				(* If no error, read one page of historical data *)
				FaultData.AlarmID 		:= ModBus.MB_Resp.Data[0];
				FaultData.SuppTime 		:= BUILD_16TO32_COPY(ModBus.MB_Resp.Data[1],ModBus.MB_Resp.Data[2]);
				FaultData.OpTime 		:= BUILD_16TO32_COPY(ModBus.MB_Resp.Data[3],ModBus.MB_Resp.Data[4]);
				FaultData.InvStatus 	:= ModBus.MB_Resp.Data[5];
				FaultData.Vpv_ref 		:= ModBus.MB_Resp.Data[6];
				FaultData.Vpv 			:= ModBus.MB_Resp.Data[7];
				FaultData.Vmain 		:= ModBus.MB_Resp.Data[8];
				FaultData.Status2 		:= ModBus.MB_Resp.Data[9];
				FaultData.Status1 		:= ModBus.MB_Resp.Data[10];
				FaultData.Tboard 		:= ModBus.MB_Resp.Data[11];
				FaultData.Tigbt 		:= ModBus.MB_Resp.Data[12];
				FaultData.I_u 			:= ModBus.MB_Resp.Data[13];
				FaultData.I_v 			:= ModBus.MB_Resp.Data[14];
				FaultData.I_w 			:= ModBus.MB_Resp.Data[15];
				FaultData.ClampStatus 	:= ModBus.MB_Resp.Data[16];
				FaultData.DigOutput 	:= ModBus.MB_Resp.Data[17];
				FaultData.IgbtFault 	:= ModBus.MB_Resp.Data[18];
				FaultData.Psupp			:= BUILD_16TO32_COPY(ModBus.MB_Resp.Data[19],ModBus.MB_Resp.Data[20]);
				FaultData.Epv 			:= BUILD_16TO32_COPY(ModBus.MB_Resp.Data[22],ModBus.MB_Resp.Data[23]);

				ModBus.MB_Lock := FALSE;		(* All 8 pages transmitted *)
				FaultAddr 	:= 0;				(* Reset start address *)
				state_fault := WAIT_STATE;
				last_state	:= WAIT_STATE;
				retry := 0;		(* Reset retry counter *)
		
			END_IF
		END_IF

	ERROR_STATE:

		IF retry>3 THEN
			IF NOT ModBus.MB_Lock THEN LogEv(EL_Alarm,EO_INV,ID,5,'');						(* ModBus not free	*)
			ELSE LogEv(EL_Alarm,EO_INV,ID,4,SEL(ModBus.MB_MASTER.MB_Error<>0,'0','1'));		(* ModBus communication error *)
			END_IF

			FaultAddr 	:= 0;
			state_fault := WAIT_STATE;
		ELSE
			retry := retry + 1;
			state_fault := last_state;
		END_IF
END_CASE
END_ACTION

(* POU Plant_Objects/obj_MODBUS_STR_ES889, ST *)
FUNCTION_BLOCK obj_MODBUS_STR_ES889
(* === MODBUS SMART STRING BOX ES889 ===
   v1.0[15/06/15] - Versioning
*)
VAR CONSTANT
		WAIT_STATE		:	BYTE := 0;
		QUERY_MEAS_1	:	BYTE := 1;
		QUERY_MEAS_2	:	BYTE := 2;
		QUERY_MASK		:	BYTE := 3;
		QUERY_PANELS	:	BYTE := 4;
		END_READ		:	BYTE := 5;

		QUERY_FAULT_LIST:	BYTE := 10;
		LOG_HISTORICAL	:	BYTE := 11;

		ERROR_STATE		:	BYTE := 100;

END_VAR
VAR_INPUT
		ID			:	BYTE;				(* Logical device ID needed for Clevergy purpose and log	*)
		Address		:	BYTE;				(* Modbus address of the device	*)

		RefreshTime	: 	TIME := T#1m;

		(* Read fault list *)
		FaultAddr	:	WORD;

		retryErrMax	:	BYTE := 15;		(* 15 minutes *)
END_VAR
VAR_IN_OUT
		ModBus		: obj_MODBUS;
END_VAR
VAR_OUTPUT
		Status_Log	: BYTE;
		Status_Vis	: DWORD;
END_VAR
VAR
		InitOK		: BOOL;			(* Flag that indicates if the VARS have been initialized or not	*)

		Data		: typ_MODBUS_STR_ES889;
		tempData	: typ_MODBUS_STR_ES889;
		FaultData	: typ_MODBUS_STR_ES889_His;

		(* Modbus State machine variables	*)
		state		:	BYTE;
		state_fault	:	BYTE;
		last_state	:	BYTE;
		retry		:	BYTE;
		retryErr	:	BYTE;
		ReadTmr		:	TON := (PT:=t#5s);
		fModbusAlr	:	BOOL;

		counter		:	BYTE;

		Alarm		: FLT_EVENT;
		WrnPerform	: FLT_EVENT;
		ModbusAlr	: FLT_EVENT := (INITEV:=FALSE);

		ActualAlarm	: BYTE;
		OldAlarm	: BYTE;
		ActualStolen: WORD;
		OldStolen	: WORD;
		OldOpen		: WORD;
		PerformWrn	: WORD;
		OldPerform	: WORD;

		AlarmCtr	: BYTE;
		WarningCtr	: BYTE;

		s1			: STRING;

		fTimeout	: BOOL;
END_VAR
IF NOT InitOK THEN
	ReadTmr.PT := WORD_TO_TIME((Plant_INV+ID)*2000);
	InitOK := TRUE;
END_IF

IF FaultAddr=0 THEN

	Stm();

	(**** Check String Box ALARM ****)
	CheckAlarm();

ELSE

	StmFault();

END_IF

(* Set "Status_Log" according to actual object status	*)
IF AlarmCtr > 0 THEN
	Status_Log := 2;
	Status_Vis := COLOR_RED;
ELSIF WarningCtr > 0 THEN
	Status_Log := 1;
	Status_Vis := COLOR_YELLOW;
ELSE
	Status_Log := 0;
	Status_Vis := COLOR_GREEN;
END_IF
END_FUNCTION_BLOCK
ACTION AddLogData:
Logger.s1:=INSERT('&STR=',BYTE_TO_STRING(ID),4);
IF ID<10 THEN Logger.s1:=INSERT(Logger.s1,'0',4); END_IF

(* Create messagge to append to the log file in string format, containing the historical value for current alarm	*)
Logger.s1:=CONCAT(Logger.s1,WORD_TO_STRING(Data.Istring1));				Logger.s1:=CONCAT(Logger.s1,';');
Logger.s1:=CONCAT(Logger.s1,WORD_TO_STRING(Data.Istring2));				Logger.s1:=CONCAT(Logger.s1,';');
Logger.s1:=CONCAT(Logger.s1,WORD_TO_STRING(Data.Istring3));				Logger.s1:=CONCAT(Logger.s1,';');
Logger.s1:=CONCAT(Logger.s1,WORD_TO_STRING(Data.Istring4));				Logger.s1:=CONCAT(Logger.s1,';');
Logger.s1:=CONCAT(Logger.s1,WORD_TO_STRING(Data.Istring5));				Logger.s1:=CONCAT(Logger.s1,';');
Logger.s1:=CONCAT(Logger.s1,WORD_TO_STRING(Data.Istring6));				Logger.s1:=CONCAT(Logger.s1,';');
Logger.s1:=CONCAT(Logger.s1,WORD_TO_STRING(Data.Istring7));				Logger.s1:=CONCAT(Logger.s1,';');
Logger.s1:=CONCAT(Logger.s1,WORD_TO_STRING(Data.Istring8));				Logger.s1:=CONCAT(Logger.s1,';');
Logger.s1:=CONCAT(Logger.s1,WORD_TO_STRING(Data.Iavg));					Logger.s1:=CONCAT(Logger.s1,';');
Logger.s1:=CONCAT(Logger.s1,WORD_TO_STRING(Data.Imax));					Logger.s1:=CONCAT(Logger.s1,';');
Logger.s1:=CONCAT(Logger.s1,WORD_TO_STRING(Data.Imin));					Logger.s1:=CONCAT(Logger.s1,';');

Logger.s1:=CONCAT(Logger.s1,INT_TO_STRING(Data.Tboard));				Logger.s1:=CONCAT(Logger.s1,';');
Logger.s1:=CONCAT(Logger.s1,INT_TO_STRING(Data.Tenv));					Logger.s1:=CONCAT(Logger.s1,';');

Logger.s1:=CONCAT(Logger.s1,WORD_TO_STRING(Data.M019));					Logger.s1:=CONCAT(Logger.s1,';');
Logger.s1:=CONCAT(Logger.s1,WORD_TO_STRING(PerformWrn));				Logger.s1:=CONCAT(Logger.s1,';');

(* Add log returned by the object	*)
Logger.s1:=CONCAT(Logger.s1,BYTE_TO_STRING(Status_Log));

(* Add the entire new string "s1" with the updated measurements to the one has to be transmitted	*)
ADDSTRING(ADR(Logger.TData), ADR(Logger.s1), Logger.TLen);
END_ACTION
ACTION AppendMeasure:
(* Used to add signifcant measurements when an alarm happens (it's a sort of historical fault list, as described at page 40
   of the Programming Manual; the only difference is that is not used the one of the string box, but it's rebuild with the
   read measurements *)
s1 := CONCAT(s1,';');
s1 := CONCAT(s1, WORD_TO_STRING(SHR(Data.M018,8)));	(* Stolen string *)
s1 := CONCAT(s1,';');
s1 := CONCAT(s1, WORD_TO_STRING(Data.M019));		(* Open string *)
s1 := CONCAT(s1,';');
s1 := CONCAT(s1, INT_TO_STRING(Data.Tboard));		(* Board temperature *)
s1 := CONCAT(s1,';');
s1 := CONCAT(s1, DWORD_TO_STRING(Data.SuppTime));	(* Supply time *)
s1 := CONCAT(s1,';');
s1 := CONCAT(s1, DWORD_TO_STRING(Data.OpTime));		(* Operation time *)
END_ACTION
ACTION CheckAlarm:
(* Verify ModBus error	*)
ModbusAlr(IN:=fModbusAlr);

IF ModbusAlr.EVH THEN
	LogEv(EL_Alarm,EO_STR,ID,4,SEL(ModBus.MB_MASTER.MB_Error<>0,'0','1'));
	AlarmCtr := AlarmCtr + 1;
END_IF

IF ModbusAlr.EVL THEN
	LogEv(EL_Log,EO_STR,ID,9,'');
	AlarmCtr := SEL(AlarmCtr=0, AlarmCtr-1, 0);
END_IF


(* Verify StringBox error/alarm	*)
ActualAlarm := WORD_TO_BYTE(Data.M018 AND 16#0F);

Alarm(IN:=(ActualAlarm <> OldAlarm));

IF Alarm.EVH THEN
	IF ActualAlarm = 0 THEN
		AlarmCtr := SEL(AlarmCtr=0, AlarmCtr-1, 0);
	ELSE
		(* Alarm codes 8 and 9 are yet checked with open and stolen string dedicated filters *)
		IF ActualAlarm<8 AND ActualAlarm>9 THEN
			LogEv(EL_Alarm,EO_STR,ID,3,BYTE_TO_STRING(ActualAlarm));
			AppendMeasure();
			AlarmCtr := AlarmCtr + 1;
		END_IF
	END_IF

	OldAlarm := ActualAlarm;
END_IF

(**** Check if another string has been stolen ****)
ActualStolen := (SHR(Data.M018,8) AND 16#00FF);

IF ActualStolen <> OldStolen THEN
	IF ActualStolen = 0 THEN
		AlarmCtr := SEL(AlarmCtr=0, AlarmCtr-1, 0);
	ELSE
		LogEv(EL_Alarm,EO_STR,ID,6,WORD_TO_STRING(ActualStolen));
		AlarmCtr := AlarmCtr + 1;
	END_IF

	OldStolen := ActualStolen;
END_IF
END_ACTION
ACTION Stm:
CASE state OF

	WAIT_STATE:	(* Refresh time manager *)

		ReadTmr(IN:=NOT(ReadTmr.Q));
		IF ReadTmr.Q THEN

			ReadTmr.PT := RefreshTime;			(* Refresh timer range *)

			(* Reset state machine variables and counters *)
			retry	:= 0;
			counter := 0;
			last_state	:= WAIT_STATE;

			(* Start state machine	*)
			state := QUERY_MEAS_1;

		END_IF


	QUERY_MEAS_1:	(* External energy counters *)
		IF NOT ModBus.MB_Start AND (NOT ModBus.MB_Lock OR retry>0) THEN
			ModBus.MB_Lock := TRUE;
			ModBus.MB_Obj := EO_STR;
			ModBus.MB_ObjId := ID;

			ModBus.MB_Query.SlaveAddress := Address;
			ModBus.MB_Query.FunctionCode := 16#3;
			ModBus.MB_Query.Read_StartAddress := 1651;
			ModBus.MB_Query.Read_Quantity := 20;
			ModBus.MB_Start := TRUE;

			state := QUERY_MEAS_2;
		END_IF

	QUERY_MEAS_2:	(* Energy supplied to the net *)

		IF NOT ModBus.MB_Start THEN
			IF ModBus.MB_MASTER.bInterfaceError<>0 OR ModBus.MB_MASTER.MB_Error<>0 THEN
				last_state := QUERY_MEAS_1;
				state := ERROR_STATE;
			ELSE

				tempData.Istring1		:= ModBus.MB_Resp.Data[0];
				tempData.Istring2		:= ModBus.MB_Resp.Data[1];
				tempData.Istring3		:= ModBus.MB_Resp.Data[2];
				tempData.Istring4		:= ModBus.MB_Resp.Data[3];
				tempData.Istring5		:= ModBus.MB_Resp.Data[4];
				tempData.Istring6		:= ModBus.MB_Resp.Data[5];
				tempData.Istring7		:= ModBus.MB_Resp.Data[6];
				tempData.Istring8		:= ModBus.MB_Resp.Data[7];
				tempData.Iavg			:= ModBus.MB_Resp.Data[8];
				tempData.Imax			:= ModBus.MB_Resp.Data[9];
				tempData.Imin			:= ModBus.MB_Resp.Data[10];

				tempData.Radiation_h	:= ModBus.MB_Resp.Data[11];
				tempData.Radiation_m	:= ModBus.MB_Resp.Data[12];
				tempData.Tmodule		:= WORD_TO_INT(ModBus.MB_Resp.Data[13]);
				tempData.Tenv			:= WORD_TO_INT(ModBus.MB_Resp.Data[14]);
				tempData.Vwind			:= ModBus.MB_Resp.Data[15];
				tempData.Tboard			:= WORD_TO_INT(ModBus.MB_Resp.Data[16]);

				tempData.M018			:= ModBus.MB_Resp.Data[17];
				tempData.M019			:= ModBus.MB_Resp.Data[18];
				tempData.M020			:= ModBus.MB_Resp.Data[19];

				ModBus.MB_Query.SlaveAddress := Address;
				ModBus.MB_Query.FunctionCode := 16#3;
				ModBus.MB_Query.Read_StartAddress := 57;
				ModBus.MB_Query.Read_Quantity := 4;
				ModBus.MB_Start := TRUE;

				state := QUERY_MASK;
			END_IF
		END_IF

	QUERY_MASK:
		IF NOT ModBus.MB_Start THEN
			IF ModBus.MB_MASTER.bInterfaceError<>0 OR ModBus.MB_MASTER.MB_Error<>0 THEN
				last_state := QUERY_MEAS_2;
				state := ERROR_STATE;
			ELSE

				tempData.SuppTime	:= BUILD_16TO32_COPY(ModBus.MB_Resp.Data[0],ModBus.MB_Resp.Data[1]);
				tempData.OpTime		:= BUILD_16TO32_COPY(ModBus.MB_Resp.Data[2],ModBus.MB_Resp.Data[3]);

				ModBus.MB_Query.SlaveAddress := Address;
				ModBus.MB_Query.FunctionCode := 16#3;
				ModBus.MB_Query.Read_StartAddress := 250;
				ModBus.MB_Query.Read_Quantity := 2;
				ModBus.MB_Start := TRUE;

				state := QUERY_PANELS;

			END_IF
		END_IF

	QUERY_PANELS:
		IF NOT ModBus.MB_Start THEN
			IF ModBus.MB_MASTER.bInterfaceError<>0 OR ModBus.MB_MASTER.MB_Error<>0 THEN
				last_state := QUERY_MASK;
				state := ERROR_STATE;
			ELSE

				tempData.Mask	:= ModBus.MB_Resp.Data[0];

				ModBus.MB_Query.SlaveAddress := Address;
				ModBus.MB_Query.FunctionCode := 16#3;
				ModBus.MB_Query.Read_StartAddress := 294;
				ModBus.MB_Query.Read_Quantity := 1;
				ModBus.MB_Start := TRUE;

				state := END_READ;

			END_IF
		END_IF

	END_READ:

		IF NOT ModBus.MB_Start THEN
			IF ModBus.MB_MASTER.bInterfaceError<>0 OR ModBus.MB_MASTER.MB_Error<>0 THEN
				last_state := QUERY_PANELS;
				state := ERROR_STATE;
			ELSE
				tempData.Panels	:= ModBus.MB_Resp.Data[0];

				(* Copy temporary data *)
				MEMCPY(ADR(tempData), ADR(Data), SIZEOF(Data));
				PerformWrn := Data.M020 AND 16#00FF;

				fModbusAlr := FALSE;
				retryErr := 0;
				ModBus.MB_Lock := FALSE;
				state := WAIT_STATE;

				(*** TEST ***)
				fTimeout := FALSE;

			END_IF
		END_IF

	ERROR_STATE:	(* Error state *)

		IF retry < 3 THEN
			retry := retry+1;
			state := last_state;

		ELSE
			ModBus.MB_Lock := FALSE;

			(* Verify if slave is dead *)
			IF retryErr < retryErrMaX THEN
				retryErr := retryErr + 1;
			ELSE
				fModbusAlr := TRUE;
			END_IF

			state := WAIT_STATE;

			(*** TEST ***)
			fTimeout := TRUE;
		END_IF


		IF ModBus.MB_MASTER.MB_Error=MB_TIME_OUT AND ID<>10 THEN
			state := state;
		END_IF
ELSE
	state := WAIT_STATE;
END_CASE
END_ACTION
ACTION StmFault:
(* State machine *)
CASE state OF

	WAIT_STATE:
		IF NOT (ModBus.MB_Lock OR ModBus.MB_Start) THEN
			ModBus.MB_Lock := TRUE;
			counter := 0;
			retry 	:= 0;
			last_state  := WAIT_STATE;
			state_fault := QUERY_FAULT_LIST;
		ELSE
			last_state  := WAIT_STATE;
			state_fault := ERROR_STATE;
		END_IF

	QUERY_FAULT_LIST:
		ModBus.MB_Query.SlaveAddress := Address;
		ModBus.MB_Query.FunctionCode := 16#3;
		ModBus.MB_Query.Read_StartAddress := FaultAddr;
		ModBus.MB_Query.Read_Quantity := 7;
		ModBus.MB_Start := TRUE;

		state := END_READ;


	END_READ:
		IF NOT ModBus.MB_Start THEN
			IF ModBus.MB_MASTER.bInterfaceError <> 0 OR ModBus.MB_MASTER.MB_Error<>0 THEN
				(* If no error, read one page of historical data *)
				FaultData.M018	 		:= ModBus.MB_Resp.Data[0];
				FaultData.M020			:= ModBus.MB_Resp.Data[1];
				FaultData.Tmodule		:= WORD_TO_INT(ModBus.MB_Resp.Data[2]);
				FaultData.SuppTime		:= BUILD_16TO32_COPY(ModBus.MB_Resp.Data[3],ModBus.MB_Resp.Data[4]);
				FaultData.OpTime		:= BUILD_16TO32_COPY(ModBus.MB_Resp.Data[5],ModBus.MB_Resp.Data[6]);


				(* Send data to server	*)
				LogEv(EL_Evt,EO_STR,ID,9,s1);

				IF counter > 7 THEN
					ModBus.MB_Lock := FALSE;		(* All 8 pages transmitted *)
					FaultAddr 	:= 0;				(* Reset start address *)
					state_fault := WAIT_STATE;
					last_state	:= WAIT_STATE;
				ELSE
					state_fault := QUERY_FAULT_LIST;
				END_IF

				retry := 0;		(* Reset retry counter *)
			ELSE
				state := ERROR_STATE;
			END_IF
		END_IF

	ERROR_STATE:

		IF retry>3 THEN
			IF NOT ModBus.MB_Lock THEN LogEv(EL_Alarm,EO_STR,ID,5,'');						(* ModBus not free	*)
			ELSE LogEv(EL_Alarm,EO_STR,ID,4,SEL(ModBus.MB_MASTER.MB_Error<>0,'0','1'));		(* ModBus communication error *)
			END_IF

			FaultAddr 	:= 0;
			state_fault := WAIT_STATE;
		ELSE
			retry := retry + 1;
			state_fault := last_state;
		END_IF
END_CASE
END_ACTION

(* POU Utils Functions/PLANT_STATUS, ST *)
FUNCTION_BLOCK PLANT_STATUS
VAR_INPUT
	obj_Status		:	WORD;
END_VAR
VAR_OUTPUT
	plantStatus		:	WORD;
END_VAR
VAR
	Pwm				:	TON := (PT:=T#1s);
END_VAR
(*CASE plantStatus OF

	0:	(* Plant OK - Everything works well *)
		Pwm(IN:=FALSE);							(* Stop timer if running *)
		LAMP_AL := FALSE;						(* Keep the lamp switched off *)

	1:	(* Plant in warning *)
		Pwm(IN:= NOT(Pwm.Q));

		IF Pwm.Q THEN
			LAMP_AL := NOT LAMP_AL;				(* Toggle output *)
		END_IF

	2:	(* Plant in alarm *)
		Pwm(IN:=FALSE);							(* Stop timer if running *)
		LAMP_AL	:= TRUE;						(* Keep the lamp switched on *)

END_CASE*)

plantStatus := 0;		(* Reset plant status *)
END_FUNCTION_BLOCK
ACTION UpdateStatus:
IF plantStatus = 2 THEN

	RETURN;					(* If plant already in alarm condition do nothing *)

ELSE
	IF obj_Status <> 0 THEN
		plantStatus := obj_Status;			(* If plant in warning/normal condition and current object in alarm, update plant status *)
	END_IF
END_IF
END_ACTION

(* POU PLC_WDT_old, ST *)
FUNCTION PLC_WDT_old: DWORD VAR_INPUT dwEvent: DWORD; dwFilter: DWORD; dwOwner: DWORD; END_VAR
LogEv(EL_AlarmStop,EO_SYS,1,10,'Watchdog');
END_FUNCTION

(* POU Utils Functions/RAW16TOHEXSTR, ST *)
FUNCTION RAW16TOHEXSTR : STRING(128)
VAR_INPUT
	pData: POINTER TO BYTE;
	DataLen: BYTE;
END_VAR
VAR
	pt: POINTER TO BYTE;
	xl: BYTE;
END_VAR
pt:=ADR(RAW16TOHEXSTR);
xl:=0;

WHILE DataLen>0 AND xl<120 DO

	pData:=pData+1;

	pt^ := (pData^ / 16#10) + 48 + (((pData^ / 16#10)/10)*7);
	pt:=pt+1;
	pt^ := (pData^ AND 16#0F)  + 48 + (((pData^ AND 16#0F)/10)*7);
	pt:=pt+1;

	pData:=pData-1;

	pt^ := (pData^ / 16#10) + 48 + (((pData^ / 16#10)/10)*7);
	pt:=pt+1;
	pt^ := (pData^ AND 16#0F)  + 48 + (((pData^ AND 16#0F)/10)*7);
	pt:=pt+1;

	xl:=xl+4;

	DataLen:=DataLen-2;
	pData:=pData+2;

END_WHILE

pt^:=0;
END_FUNCTION

(* POU Utils Functions/RAWTOHEXSTR, ST *)
FUNCTION RAWTOHEXSTR : STRING(128)
VAR_INPUT
	pData: POINTER TO BYTE;
	DataLen: BYTE;
END_VAR
VAR
	pt: POINTER TO BYTE;
	xl: BYTE;
END_VAR
pt:=ADR(RAWTOHEXSTR);

xl:=2;

WHILE DataLen>0 AND xl<128 DO

	pt^ := (pData^ / 16#10) + 48 + (((pData^ / 16#10)/10)*7);
	pt:=pt+1;
	pt^ := (pData^ AND 16#0F)  + 48 + (((pData^ AND 16#0F)/10)*7);
	pt:=pt+1;

	xl:=xl+2;

	DataLen:=DataLen-1;
	pData:=pData+1;

END_WHILE

pt^:=0;
END_FUNCTION

(* POU Utils Functions/TONOF, ST *)
FUNCTION_BLOCK TONOF
VAR_INPUT
	IN		: BOOL;
	PT_ON	: TIME; (* time to pass, before OUT is set *)
	PT_OF	: TIME; (* time to pass, before OUT is reset *)
END_VAR
VAR_OUTPUT
	OUT		: BOOL;
END_VAR
VAR
	timer	: TON;
END_VAR
IF IN<>OUT THEN
	timer(IN:=TRUE,PT:=SEL(IN,PT_OF,PT_ON));
	IF timer.Q THEN OUT:=IN; END_IF
ELSE
	timer(IN:=FALSE);
END_IF
END_FUNCTION_BLOCK

(* Visualisation PLC_VISU
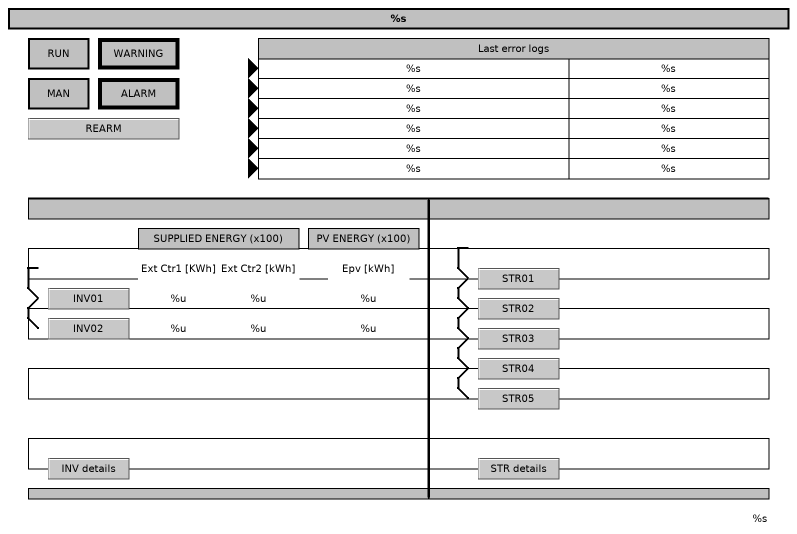
rectangle at (10,0)-(791,21): text "%s"; shows .Plant_NAME
rounded rectangle at (30,30)-(91,61): text "RUN"; alarm colour if NOT Mode_Manual; runs INTERN ASSIGN Mode_Manual:=(FALSE)
rounded rectangle at (30,70)-(91,101): text "MAN"; alarm colour if Mode_Manual; runs INTERN ASSIGN Mode_Manual:=(TRUE)
rectangle at (570,50)-(771,71): text "%s"; shows Sys.LastLogs_Msg[0]
polygon at (250,150)-(260,170): invisible if Sys.LastLogs_Idx<>0
rectangle at (570,70)-(771,91): text "%s"; shows Sys.LastLogs_Msg[1]
polygon at (250,50)-(260,70): invisible if Sys.LastLogs_Idx<>1
rectangle at (570,90)-(771,111): text "%s"; shows Sys.LastLogs_Msg[2]
polygon at (250,70)-(260,90): invisible if Sys.LastLogs_Idx<>2
rectangle at (570,110)-(771,131): text "%s"; shows Sys.LastLogs_Msg[3]
polygon at (250,90)-(260,110): invisible if Sys.LastLogs_Idx<>3
rectangle at (570,130)-(771,151): text "%s"; shows Sys.LastLogs_Msg[4]
polygon at (250,110)-(260,130): invisible if Sys.LastLogs_Idx<>4
rectangle at (570,150)-(771,171): text "%s"; shows Sys.LastLogs_Msg[5]
polygon at (250,130)-(260,150): invisible if Sys.LastLogs_Idx<>5
rectangle at (260,50)-(571,71): text "%s"; shows Sys.LastLogs_Dat[0]
rectangle at (260,70)-(571,91): text "%s"; shows Sys.LastLogs_Dat[1]
rectangle at (260,90)-(571,111): text "%s"; shows Sys.LastLogs_Dat[2]
rectangle at (260,110)-(571,131): text "%s"; shows Sys.LastLogs_Dat[3]
rectangle at (260,130)-(571,151): text "%s"; shows Sys.LastLogs_Dat[4]
rectangle at (260,150)-(571,171): text "%s"; shows Sys.LastLogs_Dat[5]
rectangle at (100,70)-(181,101): text "ALARM"; alarm colour if Sys.Alarm; runs INTERN ASSIGN Mode_Manual:=(FALSE)
rectangle at (100,30)-(181,61): text "WARNING"; alarm colour if Sys.Warning; runs INTERN ASSIGN Mode_Manual:=(TRUE)
button at (30,110)-(181,131): text "REARM"; runs INTERN ASSIGN Sys.Alarm:=(FALSE);INTERN ASSIGN Sys.Warning:=(FALSE)
button at (50,280)-(131,301): text "INV01"; runs INTERN ASSIGN INV[1].Cmd:=(0);INTERN ASSIGN INV[1].fRemoteCmd:=(TRUE)
rectangle at (260,30)-(771,51): text "Last error logs"
button at (50,310)-(131,331): text "INV02"; runs INTERN ASSIGN INV[2].Cmd:=(0);INTERN ASSIGN INV[2].fRemoteCmd:=(TRUE)
rectangle at (140,250)-(221,271): text "Ext Ctr1 [KWh]"
rectangle at (140,280)-(221,301): text "%u"; shows INV[1].Data.Esup_ExtCtr1
rectangle at (140,310)-(221,331): text "%u"; shows INV[2].Data.Esup_ExtCtr1
rounded rectangle at (140,220)-(301,241): text "SUPPLIED ENERGY (x100)"
button at (50,450)-(131,471): text "INV details"; opens PLC_VISU_INV
button at (480,260)-(561,281): text "STR01"; runs INTERN ASSIGN STR[1].Cmd:=(0);INTERN ASSIGN STR[1].fRead:=(TRUE)
button at (480,290)-(561,311): text "STR02"; runs INTERN ASSIGN STR[2].Cmd:=(0);INTERN ASSIGN STR[2].fRead:=(TRUE)
button at (480,320)-(561,341): text "STR03"; runs INTERN ASSIGN STR[3].Cmd:=(0);INTERN ASSIGN STR[3].fRead:=(TRUE)
button at (480,350)-(561,371): text "STR04"; runs INTERN ASSIGN STR[4].Cmd:=(0);INTERN ASSIGN STR[4].fRead:=(TRUE)
button at (480,380)-(561,401): text "STR05"; runs INTERN ASSIGN STR[5].Cmd:=(0);INTERN ASSIGN STR[5].fRead:=(TRUE)
button at (480,450)-(561,471): text "STR details"; opens PLC_VISU_STR
rectangle at (220,250)-(301,271): text "Ext Ctr2 [kWh]"
rectangle at (220,280)-(301,301): text "%u"; shows INV[1].Data.ExtCtr2
rectangle at (220,310)-(301,331): text "%u"; shows INV[2].Data.ExtCtr2
rounded rectangle at (310,220)-(421,241): text "PV ENERGY (x100)"
rectangle at (330,250)-(411,271): text "Epv [kWh]"
rectangle at (330,280)-(411,301): text "%u"; shows INV[1].Data.Epv
rectangle at (330,310)-(411,331): text "%u"; shows INV[2].Data.Epv
rectangle at (430,500)-(771,521): text "%s"; shows Sys.Time_LogString
15 more shapes without text or variables
9 elements of other kinds (tables, trends, ...) not read
*)

(* Visualisation PLC_VISU_INV
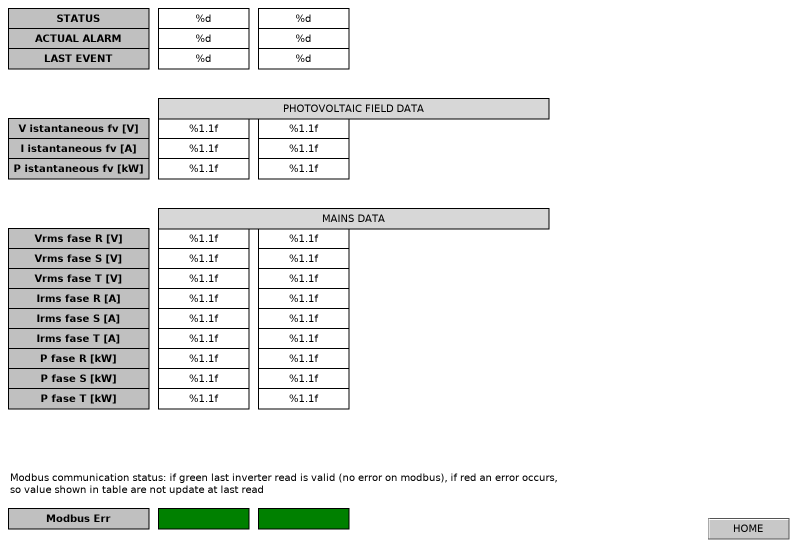
rectangle at (10,160)-(151,181): text "V istantaneous fv [V]"
rectangle at (10,180)-(151,201): text "I istantaneous fv [A]"
rectangle at (10,200)-(151,221): text "P istantaneous fv [kW]"
rectangle at (10,270)-(151,291): text "Vrms fase R [V]"
rectangle at (10,290)-(151,311): text "Vrms fase S [V]"
rectangle at (10,310)-(151,331): text "Vrms fase T [V]"
rectangle at (10,330)-(151,351): text "Irms fase R [A]"
rectangle at (10,350)-(151,371): text "Irms fase S [A]"
rectangle at (10,370)-(151,391): text "Irms fase T [A]"
rectangle at (10,390)-(151,411): text "P fase R [kW]"
rectangle at (10,410)-(151,431): text "P fase S [kW]"
rectangle at (10,430)-(151,451): text "P fase T [kW]"
rectangle at (10,50)-(151,71): text "STATUS"
rectangle at (10,70)-(151,91): text "ACTUAL ALARM"
rectangle at (160,160)-(251,181): text "%1.1f"; shows WORD_TO_REAL(.INV[1].Data.Vpv)/10
rectangle at (160,180)-(251,201): text "%1.1f"; shows WORD_TO_REAL(INV[1].Data.Ipv)/10
rectangle at (160,270)-(251,291): text "%1.1f"; shows WORD_TO_REAL(INV[1].Data.Vrms_r)/10
rectangle at (160,290)-(251,311): text "%1.1f"; shows WORD_TO_REAL(INV[1].Data.Vrms_s)/10
rectangle at (160,310)-(251,331): text "%1.1f"; shows WORD_TO_REAL(INV[1].Data.Vrms_t)/10
rectangle at (160,330)-(251,351): text "%1.1f"; shows INT_TO_REAL(INV[1].Data.Irms_r)/10
rectangle at (160,350)-(251,371): text "%1.1f"; shows INT_TO_REAL(INV[1].Data.Irms_s)/10
rectangle at (160,370)-(251,391): text "%1.1f"; shows INT_TO_REAL(INV[1].Data.Irms_t)/10
rectangle at (160,390)-(251,411): text "%1.1f"; shows INT_TO_REAL(INV[1].Data.P_r)/10
rectangle at (160,410)-(251,431): text "%1.1f"; shows INT_TO_REAL(INV[1].Data.P_s)/10
rectangle at (160,430)-(251,451): text "%1.1f"; shows INT_TO_REAL(INV[1].Data.P_t)/10
rectangle at (160,200)-(251,221): text "%1.1f"; shows INT_TO_REAL(INV[1].Data.Ppv)/10
rectangle at (160,50)-(251,71): text "%d"; shows INV[1].Data.Status
rectangle at (160,70)-(251,91): text "%d"; shows .INV[1].Data.ActiveAlarm
rectangle at (260,160)-(351,181): text "%1.1f"; shows WORD_TO_REAL(INV[2].Data.Vpv)/10
rectangle at (260,180)-(351,201): text "%1.1f"; shows WORD_TO_REAL(INV[2].Data.Ipv)/10
rectangle at (260,270)-(351,291): text "%1.1f"; shows WORD_TO_REAL(INV[2].Data.Vrms_r)/10
rectangle at (260,290)-(351,311): text "%1.1f"; shows WORD_TO_REAL(INV[2].Data.Vrms_s)/10
rectangle at (260,310)-(351,331): text "%1.1f"; shows WORD_TO_REAL(INV[2].Data.Vrms_t)/10
rectangle at (260,330)-(351,351): text "%1.1f"; shows INT_TO_REAL(INV[2].Data.Irms_r)/10
rectangle at (260,350)-(351,371): text "%1.1f"; shows INT_TO_REAL(INV[2].Data.Irms_s)/10
rectangle at (260,370)-(351,391): text "%1.1f"; shows INT_TO_REAL(INV[2].Data.Irms_t)/10
rectangle at (260,390)-(351,411): text "%1.1f"; shows INT_TO_REAL(INV[2].Data.P_r)/10
rectangle at (260,410)-(351,431): text "%1.1f"; shows INT_TO_REAL(INV[2].Data.P_s)/10
rectangle at (260,430)-(351,451): text "%1.1f"; shows INT_TO_REAL(INV[2].Data.P_t)/10
rectangle at (260,200)-(351,221): text "%1.1f"; shows INT_TO_REAL(INV[2].Data.Ppv)/10
rectangle at (260,50)-(351,71): text "%d"; shows INV[2].Data.Status
rectangle at (260,70)-(351,91): text "%d"; shows .INV[2].Data.ActiveAlarm
rounded rectangle at (160,140)-(551,161): text "PHOTOVOLTAIC FIELD DATA"
rounded rectangle at (160,250)-(551,271): text "MAINS DATA"
rectangle at (10,90)-(151,111): text "LAST EVENT"
rectangle at (160,90)-(251,111): text "%d"; shows INV[1].Data.Event
rectangle at (260,90)-(351,111): text "%d"; shows INV[2].Data.Event
button at (710,560)-(791,581): text "HOME"; opens PLC_VISU
rectangle at (10,550)-(151,571): text "Modbus Err"
rectangle at (160,550)-(251,571): alarm colour if INV[1].fTimeout
rectangle at (260,550)-(351,571): alarm colour if INV[2].fTimeout
rectangle at (10,510)-(761,541): text "Modbus communication status: if green last inverter read is valid (no error on modbus), if red an error occurs, / so value shown in table are not update at last read"
2 elements of other kinds (tables, trends, ...) not read
*)

(* Visualisation PLC_VISU_STR
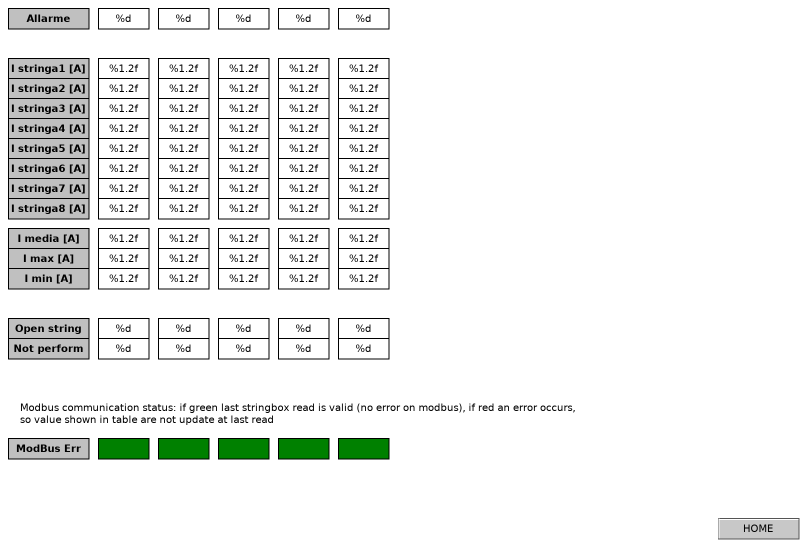
rectangle at (0,100)-(81,121): text "I stringa1 [A]"
rectangle at (0,120)-(81,141): text "I stringa2 [A]"
rectangle at (0,140)-(81,161): text "I stringa3 [A]"
rectangle at (0,160)-(81,181): text "I stringa4 [A]"
rectangle at (0,180)-(81,201): text "I stringa5 [A]"
rectangle at (90,100)-(141,121): text "%1.2f"; shows INT_TO_REAL(STR[1].Data.Istring1)/100
rectangle at (0,200)-(81,221): text "I stringa6 [A]"
rectangle at (0,220)-(81,241): text "I stringa7 [A]"
rectangle at (0,240)-(81,261): text "I stringa8 [A]"
rectangle at (0,270)-(81,291): text "I media [A]"
rectangle at (0,290)-(81,311): text "I max [A]"
rectangle at (0,310)-(81,331): text "I min [A]"
rectangle at (0,50)-(81,71): text "Allarme"
rectangle at (90,50)-(141,71): text "%d"; shows .STR[1].ActualAlarm
rectangle at (90,120)-(141,141): text "%1.2f"; shows INT_TO_REAL(STR[1].Data.Istring2)/100
rectangle at (90,140)-(141,161): text "%1.2f"; shows INT_TO_REAL(STR[1].Data.Istring3)/100
rectangle at (90,160)-(141,181): text "%1.2f"; shows INT_TO_REAL(STR[1].Data.Istring4)/100
rectangle at (90,180)-(141,201): text "%1.2f"; shows INT_TO_REAL(STR[1].Data.Istring5)/100
rectangle at (90,200)-(141,221): text "%1.2f"; shows INT_TO_REAL(STR[1].Data.Istring6)/100
rectangle at (90,220)-(141,241): text "%1.2f"; shows INT_TO_REAL(STR[1].Data.Istring7)/100
rectangle at (90,240)-(141,261): text "%1.2f"; shows INT_TO_REAL(STR[1].Data.Istring8)/100
rectangle at (90,270)-(141,291): text "%1.2f"; shows INT_TO_REAL(STR[1].Data.Iavg)/100
rectangle at (90,290)-(141,311): text "%1.2f"; shows INT_TO_REAL(STR[1].Data.Imax)/100
rectangle at (90,310)-(141,331): text "%1.2f"; shows INT_TO_REAL(STR[1].Data.Imin)/100
rectangle at (150,100)-(201,121): text "%1.2f"; shows INT_TO_REAL(STR[2].Data.Istring1)/100
rectangle at (150,50)-(201,71): text "%d"; shows .STR[2].ActualAlarm
rectangle at (150,120)-(201,141): text "%1.2f"; shows INT_TO_REAL(STR[2].Data.Istring2)/100
rectangle at (150,140)-(201,161): text "%1.2f"; shows INT_TO_REAL(STR[2].Data.Istring3)/100
rectangle at (150,160)-(201,181): text "%1.2f"; shows INT_TO_REAL(STR[2].Data.Istring4)/100
rectangle at (150,180)-(201,201): text "%1.2f"; shows INT_TO_REAL(STR[2].Data.Istring5)/100
rectangle at (150,200)-(201,221): text "%1.2f"; shows INT_TO_REAL(STR[2].Data.Istring6)/100
rectangle at (150,220)-(201,241): text "%1.2f"; shows INT_TO_REAL(STR[2].Data.Istring7)/100
rectangle at (150,240)-(201,261): text "%1.2f"; shows INT_TO_REAL(STR[2].Data.Istring8)/100
rectangle at (150,270)-(201,291): text "%1.2f"; shows INT_TO_REAL(STR[2].Data.Iavg)/100
rectangle at (150,290)-(201,311): text "%1.2f"; shows INT_TO_REAL(STR[2].Data.Imax)/100
rectangle at (150,310)-(201,331): text "%1.2f"; shows INT_TO_REAL(STR[2].Data.Imin)/100
rectangle at (210,100)-(261,121): text "%1.2f"; shows INT_TO_REAL(STR[3].Data.Istring1)/100
rectangle at (210,50)-(261,71): text "%d"; shows .STR[3].ActualAlarm
rectangle at (210,120)-(261,141): text "%1.2f"; shows INT_TO_REAL(STR[3].Data.Istring2)/100
rectangle at (210,140)-(261,161): text "%1.2f"; shows INT_TO_REAL(STR[3].Data.Istring3)/100
rectangle at (210,160)-(261,181): text "%1.2f"; shows INT_TO_REAL(STR[3].Data.Istring4)/100
rectangle at (210,180)-(261,201): text "%1.2f"; shows INT_TO_REAL(STR[3].Data.Istring5)/100
rectangle at (210,200)-(261,221): text "%1.2f"; shows INT_TO_REAL(STR[3].Data.Istring6)/100
rectangle at (210,220)-(261,241): text "%1.2f"; shows INT_TO_REAL(STR[3].Data.Istring7)/100
rectangle at (210,240)-(261,261): text "%1.2f"; shows INT_TO_REAL(STR[3].Data.Istring8)/100
rectangle at (210,270)-(261,291): text "%1.2f"; shows INT_TO_REAL(STR[3].Data.Iavg)/100
rectangle at (210,290)-(261,311): text "%1.2f"; shows INT_TO_REAL(STR[3].Data.Imax)/100
rectangle at (210,310)-(261,331): text "%1.2f"; shows INT_TO_REAL(STR[3].Data.Imin)/100
rectangle at (270,100)-(321,121): text "%1.2f"; shows INT_TO_REAL(STR[4].Data.Istring1)/100
rectangle at (270,50)-(321,71): text "%d"; shows .STR[4].ActualAlarm
rectangle at (270,120)-(321,141): text "%1.2f"; shows INT_TO_REAL(STR[4].Data.Istring2)/100
rectangle at (270,140)-(321,161): text "%1.2f"; shows INT_TO_REAL(STR[4].Data.Istring3)/100
rectangle at (270,160)-(321,181): text "%1.2f"; shows INT_TO_REAL(STR[4].Data.Istring4)/100
rectangle at (270,180)-(321,201): text "%1.2f"; shows INT_TO_REAL(STR[4].Data.Istring5)/100
rectangle at (270,200)-(321,221): text "%1.2f"; shows INT_TO_REAL(STR[4].Data.Istring6)/100
rectangle at (270,220)-(321,241): text "%1.2f"; shows INT_TO_REAL(STR[4].Data.Istring7)/100
rectangle at (270,240)-(321,261): text "%1.2f"; shows INT_TO_REAL(STR[4].Data.Istring8)/100
rectangle at (270,270)-(321,291): text "%1.2f"; shows INT_TO_REAL(STR[4].Data.Iavg)/100
rectangle at (270,290)-(321,311): text "%1.2f"; shows INT_TO_REAL(STR[4].Data.Imax)/100
rectangle at (270,310)-(321,331): text "%1.2f"; shows INT_TO_REAL(STR[4].Data.Imin)/100
rectangle at (330,100)-(381,121): text "%1.2f"; shows INT_TO_REAL(STR[5].Data.Istring1)/100
rectangle at (330,50)-(381,71): text "%d"; shows .STR[5].ActualAlarm
rectangle at (330,120)-(381,141): text "%1.2f"; shows INT_TO_REAL(STR[5].Data.Istring2)/100
rectangle at (330,140)-(381,161): text "%1.2f"; shows INT_TO_REAL(STR[5].Data.Istring3)/100
rectangle at (330,160)-(381,181): text "%1.2f"; shows INT_TO_REAL(STR[5].Data.Istring4)/100
rectangle at (330,180)-(381,201): text "%1.2f"; shows INT_TO_REAL(STR[5].Data.Istring5)/100
rectangle at (330,200)-(381,221): text "%1.2f"; shows INT_TO_REAL(STR[5].Data.Istring6)/100
rectangle at (330,220)-(381,241): text "%1.2f"; shows INT_TO_REAL(STR[5].Data.Istring7)/100
rectangle at (330,240)-(381,261): text "%1.2f"; shows INT_TO_REAL(STR[5].Data.Istring8)/100
rectangle at (330,270)-(381,291): text "%1.2f"; shows INT_TO_REAL(STR[5].Data.Iavg)/100
rectangle at (330,290)-(381,311): text "%1.2f"; shows INT_TO_REAL(STR[5].Data.Imax)/100
rectangle at (330,310)-(381,331): text "%1.2f"; shows INT_TO_REAL(STR[5].Data.Imin)/100
button at (710,560)-(791,581): text "HOME"; opens PLC_VISU
rectangle at (0,480)-(81,501): text "ModBus Err"
rectangle at (90,480)-(141,501): alarm colour if STR[1].fTimeout
rectangle at (0,360)-(81,381): text "Open string"
rectangle at (90,360)-(141,381): text "%d"; shows STR[1].Data.M019
rectangle at (150,360)-(201,381): text "%d"; shows STR[2].Data.M019
rectangle at (210,360)-(261,381): text "%d"; shows STR[3].Data.M019
rectangle at (270,360)-(321,381): text "%d"; shows STR[4].Data.M019
rectangle at (330,360)-(381,381): text "%d"; shows STR[5].Data.M019
rectangle at (0,380)-(81,401): text "Not perform"
rectangle at (90,380)-(141,401): text "%d"; shows STR[1].PerformWrn
rectangle at (150,380)-(201,401): text "%d"; shows STR[2].PerformWrn
rectangle at (210,380)-(261,401): text "%d"; shows STR[3].PerformWrn
rectangle at (270,380)-(321,401): text "%d"; shows STR[4].PerformWrn
rectangle at (330,380)-(381,401): text "%d"; shows STR[5].PerformWrn
rectangle at (150,480)-(201,501): alarm colour if STR[2].fTimeout
rectangle at (210,480)-(261,501): alarm colour if STR[3].fTimeout
rectangle at (270,480)-(321,501): alarm colour if STR[4].fTimeout
rectangle at (330,480)-(381,501): alarm colour if STR[5].fTimeout
rectangle at (10,440)-(761,471): text "Modbus communication status: if green last stringbox read is valid (no error on modbus), if red an error occurs, / so value shown in table are not update at last read"
5 elements of other kinds (tables, trends, ...) not read
*)
